(* PLC project Addition_LD, IEC61131-3 LD Demo Project LD Addition Example 1.0 *)
(* stored: creationDateTime 2026-01-18T00:00:00, contentDescription LD梯形图加法示例程序 - 教学演示用, modificationDateTime 2026-01-18T00:00:00 *)

(* <h2>LD梯形图加法示例程序</h2> <p><strong>功能</strong>：实现两个INT类型整数的加法运算</p> <p><strong>变量</strong>：</p> <ul> <li>A (INT)：加数1，范围 -32768 到 32767</li> <li>B (INT)：加数2，范围 -32768 到 32767</li> <li>Result (INT)：和，存储计算结果</li> </ul> <p><strong>逻辑</strong>：使用标准ADD功能块实现 Result = A + B</p> <p><strong>测试用例</strong>：参见 examples/ld/test-cases.json</p> <p><strong>使用指南</strong>：参见 examples/ld/addition.md</p> *)
PROGRAM Addition_LD
  VAR
    A : INT;  (* 加数1：INT类型（16位有符号整数），范围 -32768 到 32767 *)
    B : INT;  (* 加数2：INT类型（16位有符号整数），范围 -32768 到 32767 *)
    Result : INT;  (* 和：存储A + B的计算结果（INT类型，可能发生溢出回绕） *)
  END_VAR

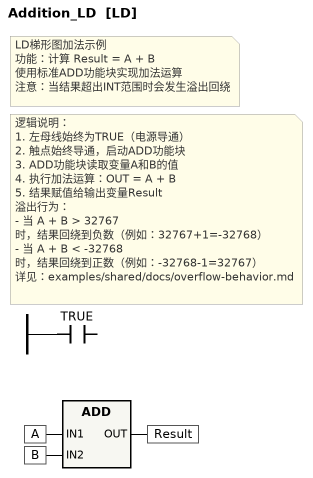
(* LD diagram, written out as Structured Text *)
(* LD梯形图加法示例
                  功能：计算 Result = A + B
                  使用标准ADD功能块实现加法运算
                  注意：当结果超出INT范围时会发生溢出回绕 *)
Result := A + B;
(* 逻辑说明：
                  1. 左母线始终为TRUE（电源导通）
                  2. 触点始终导通，启动ADD功能块
                  3. ADD功能块读取变量A和B的值
                  4. 执行加法运算：OUT = A + B
                  5. 结果赋值给输出变量Result

                  溢出行为：
                  - 当 A + B > 32767 时，结果回绕到负数（例如：32767+1=-32768）
                  - 当 A + B < -32768 时，结果回绕到正数（例如：-32768-1=32767）
                  详见：examples/shared/docs/overflow-behavior.md *)
(* drawn but not wired to any output: TRUE *)
END_PROGRAM

CONFIGURATION Config
  RESOURCE Resource1 ON PLC
    TASK MainTask(INTERVAL := T#100ms, PRIORITY := 0);
    PROGRAM Addition_LD_Instance WITH MainTask : Addition_LD;
  END_RESOURCE
END_CONFIGURATION
